{attribute 'linkalways'} 
{attribute 'no_explicit_call' := 'This FB is a CLASS and must be accessed using methods or properties'}
{attribute 'enable_dynamic_creation'}
FUNCTION_BLOCK Node_RGBA_MAGENTA EXTENDS VisionNode
VAR
    out : _TcVnVector4_LREAL;
END_VAR

METHOD PUBLIC  Clone : I_Node
VAR
	pNode : POINTER TO Node_RGBA_MAGENTA;
END_VAR
pNode := __NEW(Node_RGBA_MAGENTA);
Clone := pNode^;
END_METHOD

METHOD FB_init : BOOL
VAR_INPUT
	bInitRetains : BOOL; // if TRUE, the retain variables are initialized (warm start / cold start)
	bInCopyCode : BOOL;  // if TRUE, the instance afterwards gets moved into the copy code (online change)
END_VAR
AddOutput('out', out);
END_METHOD

METHOD PROTECTED OnExecute : HRESULT
out.Value := GVL_COLOURS.RGBA_MAGENTA;
END_METHOD

METHOD PUBLIC PreExecutionCheck
VAR_INPUT
	Check : I_PreExecutionChecks;
END_VAR
END_METHOD

END_FUNCTION_BLOCK

(* stored: Version 1.1.0.1, ProductVersion 3.1.4024.13
   POU Node_RGBA_MAGENTA: Id {55d7b74f-e302-0fc5-38a8-7da0f40f32ae}, SpecialFunc None
   Folder Constructor: Id {e126b64c-ae13-04e7-20a2-abb334d66e88}
   Method Clone: Id {e18ff29c-1613-0810-0cc7-4383df63e789}
   Method FB_init: Id {a4c62969-8240-0be5-146d-a242ace86830}
   Method OnExecute: Id {f58b7155-fc87-0485-260b-388d320dd95b}
   Method PreExecutionCheck: Id {cb845289-bf2c-02d1-0cdb-4084561d27bd} *)
